// Mitsubishi GX Works2 project: JuiceProject221129   PLC: FX3G

// global labels: Global1
VAR_GLOBAL
  orange_stock AT D1106 : REAL;  (* רגיסטר מלאי תפוזים *)
  pomelo_stock AT D1108 : REAL;  (* רגיסטר מלאי פומלות *)
  clementine_stock AT D1110 : REAL;  (* רגיסטר מלאי קלמנטינות *)
  orange_washing AT D1112 : REAL;  (* רגיסטר מכונת שטיפה תפוזים *)
  pomelo_washing AT D1114 : REAL;  (* רגיסטר מכונת שטיפה פומלות *)
  clementine_washing AT D1116 : REAL;  (* רגיסטר מכונת שטיפה קלמנטינות *)
  squeeze_container AT D1124 : REAL;  (* מיכל סחיטה *)
  juice_container AT D1126 : REAL;  (* מיכל מיץ *)
  analog_input_2 AT D8281 : INT;  (* בדיקת איכות באמצעות ערך אנלוגי 2 *)
  storage_container AT D1128 : REAL;  (* מיכל אחסון *)
  start_wash_SW AT X002 : BOOL;  (* מתג תחילת תהליך השטיפה *)
  timer0 AT TC0 : BOOL;  (* טיימר הדלקת נורה *)
  var_time_0 AT D1130 : INT;  (* זמן הדלקת נורה לטיימר 0 *)
  start_light_help AT M0 : BOOL;  (* נורת עזר לתחילת טיימר הדלקת נורה *)
  timer0_ans AT TS0 : BOOL;  (* תשובה לטיימר 0 *)
  starter_wash_help AT M1 : BOOL;  (* נורת עזר המתחילה את תהליך הדלקת הנורה *)
  switch_2 AT X002 : BOOL;  (* מתג הפעלת שטיפת פירות *)
  light_5 AT Y005 : BOOL;  (* הדלקת נורה לתחילת השטיפה *)
  start_collect AT X001 : BOOL;  (* תחילת איסוף הפירות *)
  light_1 AT Y001 : BOOL;  (* נורת איסוף פירות *)
  start_sqeeze_help AT M3 : BOOL;  (* נורת עזר לתחילת שלב הסחיטה *)
END_VAR
VAR_GLOBAL CONSTANT
  const300 : INT := 30;  (* קבוע 3 שניות *)
END_VAR
VAR_GLOBAL
  start_func1_help AT M4 : BOOL;  (* מפעיל פונקציית שטיפה *)
  holder_m1 AT M1 : BOOL;  (* מפעיל פונקציית שטיפה *)
  start_sqeeze AT X011 : BOOL;  (* תחילת שלב הסחיטה *)
  counter1 AT CC1 : BOOL;  (* מונה לחיצות על X11 *)
END_VAR
VAR_GLOBAL CONSTANT
  var_count1 : INT := 2;  (* קבוע טיימר משתנה *)
END_VAR
VAR_GLOBAL
  counter1_ans AT CS1 : BOOL;  (* תשובה למונה 1 *)
  timer2_ans AT TS2 : BOOL;  (* תשובה למונה 2 *)
  helper_blink_cycle AT M5 : BOOL;  (* נורת עזר למעגל הבהוב *)
  timer4_ans AT TS4 : BOOL;  (* תשובה לטיימר 4 *)
END_VAR
VAR_GLOBAL CONSTANT
  const50 : INT := 50;  (* קבוע 5 שניות *)
END_VAR
VAR_GLOBAL
  light_blink_helper6 AT M6 : BOOL;  (* נורת עזר להבהוב 1 *)
  timer2 AT TC2 : BOOL;  (* מונה 2 *)
  timer3 AT TC3 : BOOL;  (* מונה 3 *)
  timer3_ans AT TS3 : BOOL;  (* תשובה למונה 3 *)
  light_blink_helper7 AT M7 : BOOL;  (* נורת עזר להבהוב 2 *)
  timer4 AT TC4 : BOOL;  (* טיימר 4 *)
  light_blink_helper8 AT M8 : BOOL;  (* נורת עזר להעברה למיכל המיץ *)
  start_QA AT X003 : BOOL;  (* תחילת בדיקת איכות *)
  start_QA_help AT M9 : BOOL;  (* נורת עזר לבדיקת איכות *)
END_VAR
VAR_GLOBAL CONSTANT
  min_value_QA : REAL := 1.0;  (* ערך מינמלי לבדיקת איכות *)
END_VAR
VAR_GLOBAL
  min_val_help AT M11 : BOOL;  (* נורת עזר לבדיקת מינימום *)
END_VAR
VAR_GLOBAL CONSTANT
  max_val1 : REAL := 5.0;  (* ערך מקסימלי לבדיקת איכות *)
END_VAR
VAR_GLOBAL
  max_val_help AT M12 : BOOL;  (* נורת עזר לבדיקת מקסימום *)
  QA_sample1 AT D1134 : REAL;  (* דגימת איכות לאחר המרה *)
  check_help AT M10 : BOOL;  (* נורת עזר להפעלת בדיקת איכות *)
  QA_sample AT D1132 : INT;  (* דגימת איכות *)
END_VAR
VAR_GLOBAL CONSTANT
  k_div : REAL := 404.5;  (* קבוע חלוקה *)
END_VAR
VAR_GLOBAL
  QA_correct AT M13 : BOOL;  (* נורת עזר לבדיקת מקסימום *)
  timer5 AT TC5 : BOOL;  (* טיימר 5 *)
END_VAR
VAR_GLOBAL CONSTANT
  const5 : INT := 5;  (* קבוע 5 שניות *)
END_VAR
VAR_GLOBAL
  timer5_ans AT TS5 : BOOL;  (* תשובה לטיי מר5 *)
  QA_light_helper14 AT M14 : BOOL;  (* נורת עזר להדלקת נורת איכות *)
  counter2 AT CC2 : BOOL;  (* מונה למספר בדיקות איכות באיטרציה *)
  counter2_ans AT CS2 : BOOL;  (* תשובה למונה 2 *)
  reset_light_help15 AT M15 : BOOL;  (* נורת עזר לאיפוס *)
END_VAR
VAR_GLOBAL CONSTANT
  const500 : INT := 50;  (* קבוע 5 שניות *)
END_VAR
VAR_GLOBAL
  holder_timer_QA AT M16 : BOOL;  (* נורת עזר להחזקת הטיימר לנורת בדיקת איכות *)
  light_4 AT Y004 : BOOL;  (* נורת בדיקת איכות *)
  finish_QA_help AT M17 : BOOL;  (* נורת עזר לאינדיקציה לסיום בדיקת איכות *)
  QA_failed_help AT M18 : BOOL;  (* נורת עזר לאינדיקציה לכשלון בדיקת האיכות *)
  switch_10_startDay AT X010 : BOOL;  (* מתג תחילת יום *)
  light_10_while_work AT Y010 : BOOL;  (* נורת יום עבודה פעיל *)
  finish_day19_help AT M19 : BOOL;  (* נורת עזר לאינדיקציה לסיום יום *)
END_VAR
VAR_GLOBAL CONSTANT
  const2 : REAL := 2.0;  (* קבוע 2 שנית *)
END_VAR
VAR_GLOBAL
  pomelo_right_help20 AT M20 : BOOL;  (* נורת עזר לעמידה בתנאי תחילת יום *)
  con_start_day_help21 AT M21 : BOOL;  (* נורת עזר לעמידה בתנאי תחילת יום *)
END_VAR
VAR_GLOBAL CONSTANT
  const100 : REAL := 100.0;  (* קבוע 100 *)
END_VAR
VAR_GLOBAL
  orange_allowed AT D1136 : REAL;  (* רגיסטר השומר כמה תפוזים ניקח באיטרציה *)
  clementine_allowed AT D1138 : REAL;  (* רגיסטר השומר כמה קלמנטיות ניקח באיטרציה *)
  switch_end_day7 AT X007 : BOOL;  (* מתג חירום לסיום יום עבודה *)
  finish_iteration_help AT M22 : BOOL;  (* נורת עזר לאינדיקציה לסיום איטרציה *)
  finish_iteration_help2 AT M23 : BOOL;  (* נורת עזר לאינדיקציה לסיום איטרציה *)
  inventory_ends AT M24 : BOOL;  (* נורת עזר לבדיקת מצב המלאי בסיום איטרציה *)
END_VAR
VAR_GLOBAL CONSTANT
  const0 : REAL;  (* קבוע 0 *)
END_VAR
VAR_GLOBAL
  start_blink_help_25 AT M25 : BOOL;  (* תחילת הבהוה נורות גנרי *)
  light_2 AT Y002 : BOOL;  (* נורת סחיטה Y2 *)
  light_3 AT Y003 : BOOL;  (* נורת סחיטה Y3 *)
  light_26_help AT M26 : BOOL;  (* נורת עזר להבהוב *)
  light_blink_end_help_26 AT M26 : BOOL;  (* נורת עזר להפעלת הבהוב סוף יום *)
  light_help_27 AT M27 : BOOL;  (* נורת עזר להפעלת הבהוב סוף יום *)
  temp AT X005 : BOOL;
  timer6 AT TC6 : BOOL;  (* טיימר 6 *)
  timer6_ans AT TS6 : BOOL;  (* תשובה לטיימר6 *)
  finish_iteration_forever_help AT M30 : BOOL;  (* טיימר הדלקת נורה *)
  rst_OA_help AT M28 : BOOL;  (* נורת עזר לאיפוס בדיקת איכות *)
  finish_rst_inv29 AT M29 : BOOL;  (* נורת עזר לאינדיקציה לסיום איפוס משתני מלאי סוף יום *)
  while_day_help31 AT M31 : BOOL;
  timer7 AT TC7 : BOOL;  (* טיימר הדלקת נורה *)
  Timer7_ans AT TS7 : BOOL;  (* תשובה למונה7 *)
  analog_output_2 AT D8282 : INT;  (* יציאת ערך אנלוגי 2 *)
END_VAR
VAR_GLOBAL CONSTANT
  const00 : INT;  (* קבוע 0 *)
END_VAR
VAR_GLOBAL
  helper_start_day_34 AT M34 : BOOL;  (* נורת עזר לאינדיקציה על סיום איפוס הרגיסטרים בתחילת יום *)
  orange_passed_help_35 AT M35 : BOOL;  (* נורת עזר לאינדיקציה על סיום איפוס הרגיסטרים בתחילת יום *)
  temp1000 AT M100 : BOOL;
  dounation_time_help32 AT M32 : BOOL;  (* נורת עזר לאינדיקציה לסיום יום *)
END_VAR
VAR_GLOBAL CONSTANT
  const_dounation : REAL := 300.0;  (* קבוע לגובה המלאי לצורך תרומה *)
END_VAR
VAR_GLOBAL
  dounation_allowed33 AT M33 : BOOL;  (* נורת עזר לאינדיקציה לביצוע תרומה *)
END_VAR
VAR_GLOBAL CONSTANT
  const_dounation_prec : REAL := 0.5;  (* קבוע אחוז התרומה *)
END_VAR
VAR_GLOBAL
  timer8 AT TC8 : BOOL;  (* טיימר הדלקת נורה *)
  timer8_ans AT TS8 : BOOL;  (* תשובה לטיימר סעיף יצירתי *)
  orange_full_stock AT D1100 : REAL;  (* רגיסטר מלאי תחילת יום תפוזים *)
  pomelo_full_stock AT D1102 : REAL;  (* רגיסטר מלאי תחילת יום פומלות *)
  clementine_full_stock AT D1104 : REAL;  (* רגיסטר מלאי תחילת יום קלמנטינות *)
  light7_dounation AT Y007 : BOOL;  (* נורת תרומה *)
  temp_36 AT M36 : BOOL;  (* נורת עזר לתרומה *)
  counter3 AT CC3 : BOOL;  (* מעיד על יום עבודה *)
  counter3_ans AT CS3 : BOOL;  (* תשובה למונה 3 *)
  temp37 AT M37 : BOOL;
  temp_38 AT M38 : BOOL;
END_VAR
VAR_GLOBAL CONSTANT
  resftyfty : BOOL := 1;  (* תשובה למונה 3 *)
END_VAR
VAR_GLOBAL
  analog_output_help AT D8282 : REAL;  (* יציאת ערך אנלוגי 2 *)
  timer9 AT TC9 : BOOL;  (* טיימר הדלקת נורה *)
  timer9_ans AT TS9 : BOOL;  (* טיימר הדלקת נורה *)
  clemantino_right_help40 AT M40 : BOOL;
  inventory_ends_help41 AT M41 : BOOL;  (* נורת עזר לסיום מלאי *)
  timer10 AT TC10 : BOOL;  (* טיימר הדלקת נורה *)
  Timer10_ans AT TS10 : BOOL;  (* תשובה למונה10 *)
  temp42 AT M42 : BOOL;
  finsh_collect_help AT M100 : BOOL;  (* נורת עזר לסיום איסוף *)
END_VAR

// task Task_01 (event TRUE, interval 0, priority 31): POU_01

PROGRAM POU_01
VAR
  TC5 : BOOL;  (* תשובה למונה 1 *)
END_VAR
(* structured ladder/FBD written out as ST: instructions are called as NAME(EN, inputs, outputs); _pN, _eN, _tN stand for wires *)
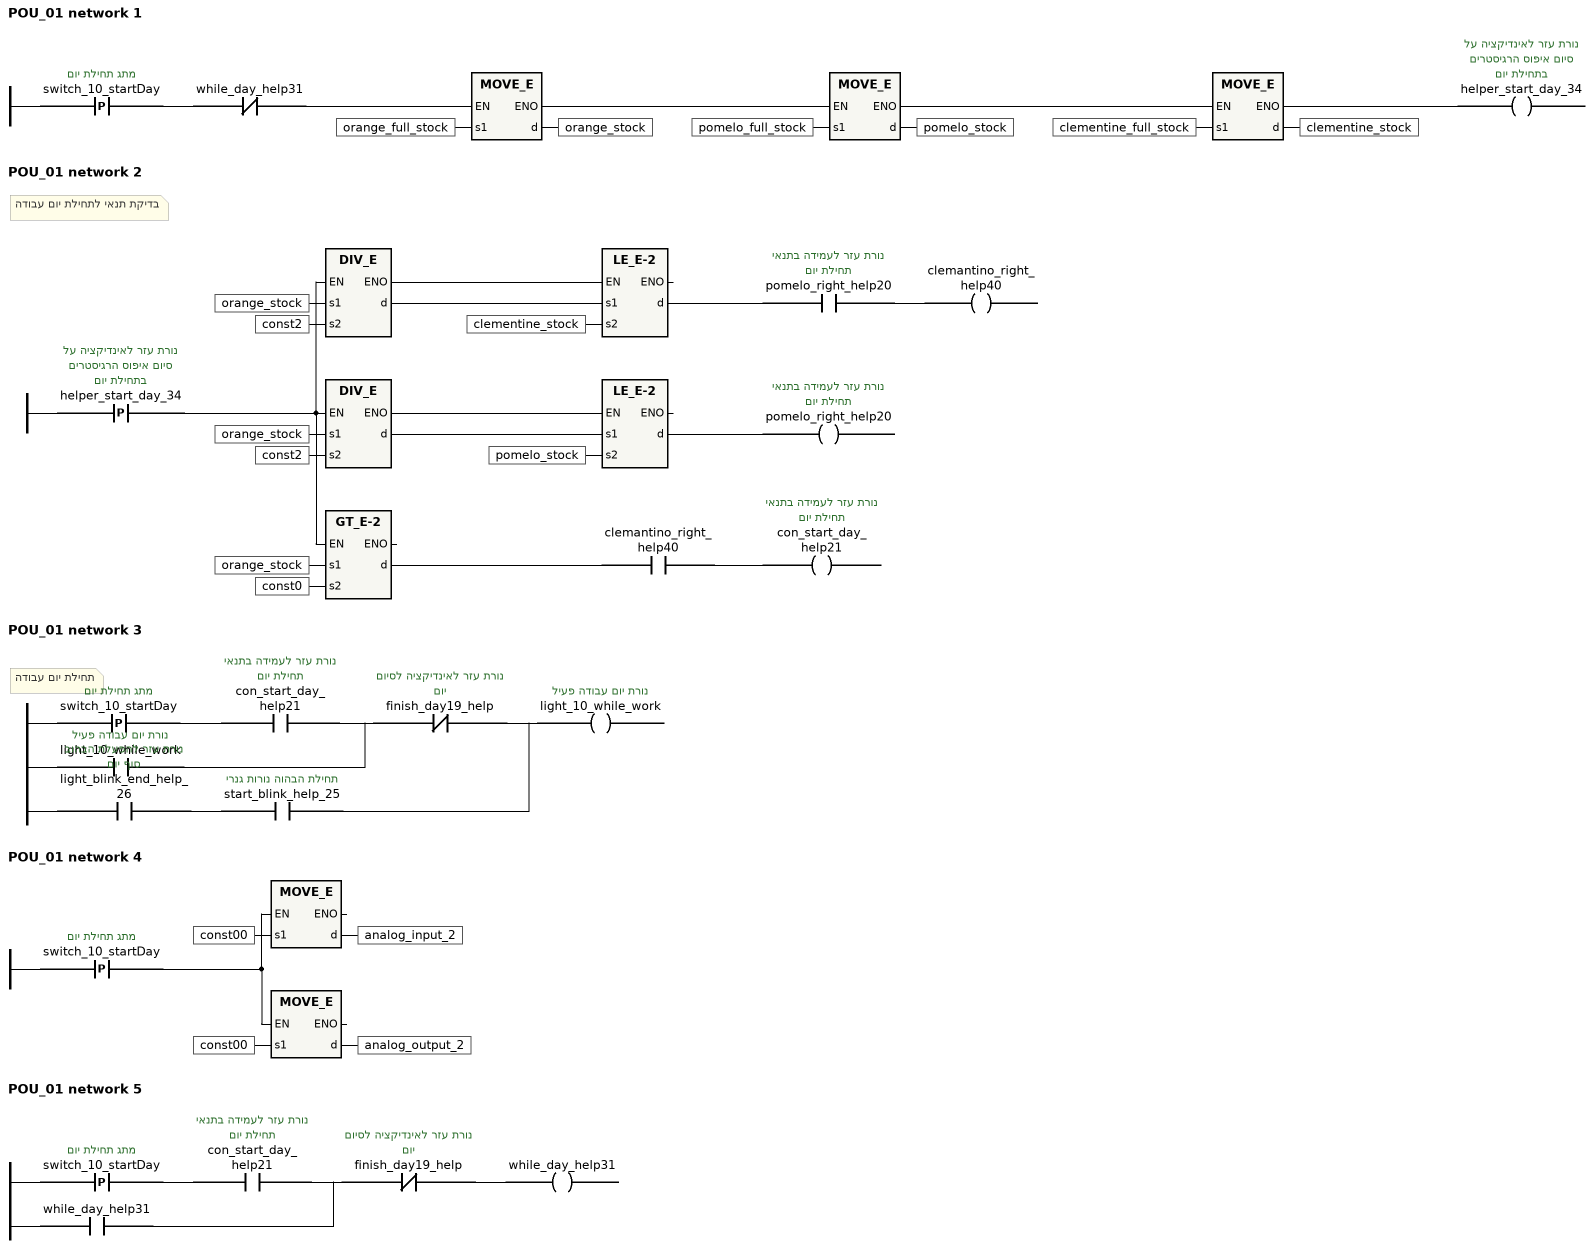
(* network 1 *)
_e1 := MOVE_E(LDP(TRUE, switch_10_startDay) AND NOT while_day_help31, orange_full_stock, orange_stock);
_e2 := MOVE_E(_e1, pomelo_full_stock, pomelo_stock);
_e3 := MOVE_E(_e2, clementine_full_stock, clementine_stock);
helper_start_day_34 := _e3;
(* network 2 *)
(* בדיקת תנאי לתחילת יום עבודה *)
_p1 := LDP(TRUE, helper_start_day_34);
_e3 := DIV_E(_p1, orange_stock, const2, _t2);
LE_E(_e3, _t2, pomelo_stock, _t4);
pomelo_right_help20 := _t4;
_e6 := DIV_E(_p1, orange_stock, const2, _t5);
LE_E(_e6, _t5, clementine_stock, _t7);
clemantino_right_help40 := _t7 AND pomelo_right_help20;
GT_E(_p1, orange_stock, const0, _t8);
con_start_day_help21 := _t8 AND clemantino_right_help40;
(* network 3 *)
(* תחילת יום עבודה *)
light_10_while_work := (((LDP(TRUE, switch_10_startDay) AND con_start_day_help21) OR light_10_while_work) AND NOT finish_day19_help) OR (light_blink_end_help_26 AND start_blink_help_25);
(* network 4 *)
_p1 := LDP(TRUE, switch_10_startDay);
MOVE_E(_p1, const00, analog_input_2);
MOVE_E(_p1, const00, analog_output_2);
(* network 5 *)
while_day_help31 := ((LDP(TRUE, switch_10_startDay) AND con_start_day_help21) OR while_day_help31) AND NOT finish_day19_help;
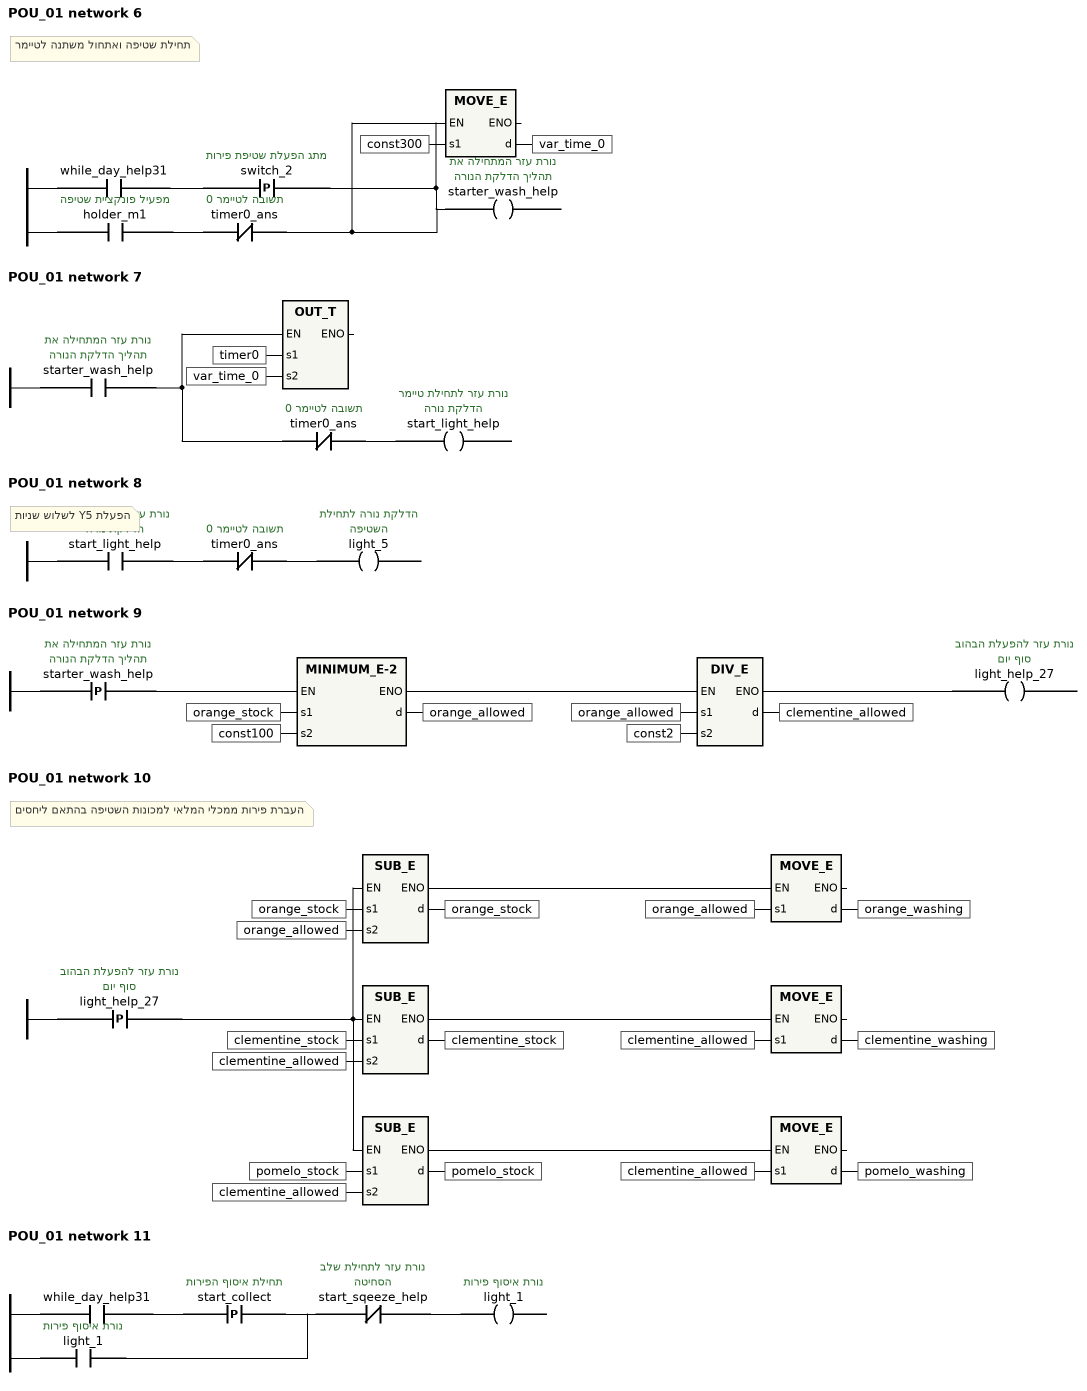
(* network 6 *)
(* תחילת שטיפה ואתחול משתנה לטיימר *)
_p1 := (while_day_help31 AND LDP(TRUE, switch_2)) OR (holder_m1 AND NOT timer0_ans);
MOVE_E(_p1, const300, var_time_0);
starter_wash_help := _p1;
(* network 7 *)
OUT_T(starter_wash_help, timer0, var_time_0);
start_light_help := starter_wash_help AND NOT timer0_ans;
(* network 8 *)
(* הפעלת Y5 לשלוש שניות *)
light_5 := start_light_help AND NOT timer0_ans;
(* network 9 *)
_e1 := MINIMUM_E(LDP(TRUE, starter_wash_help), orange_stock, const100, orange_allowed);
_e2 := DIV_E(_e1, orange_allowed, const2, clementine_allowed);
light_help_27 := _e2;
(* network 10 *)
(* העברת פירות ממכלי המלאי למכונות השטיפה בהתאם ליחסים *)
_p1 := LDP(TRUE, light_help_27);
_e2 := SUB_E(_p1, orange_stock, orange_allowed, orange_stock);
MOVE_E(_e2, orange_allowed, orange_washing);
_e3 := SUB_E(_p1, clementine_stock, clementine_allowed, clementine_stock);
MOVE_E(_e3, clementine_allowed, clementine_washing);
_e4 := SUB_E(_p1, pomelo_stock, clementine_allowed, pomelo_stock);
MOVE_E(_e4, clementine_allowed, pomelo_washing);
(* network 11 *)
light_1 := ((while_day_help31 AND LDP(TRUE, start_collect)) OR light_1) AND NOT start_sqeeze_help;
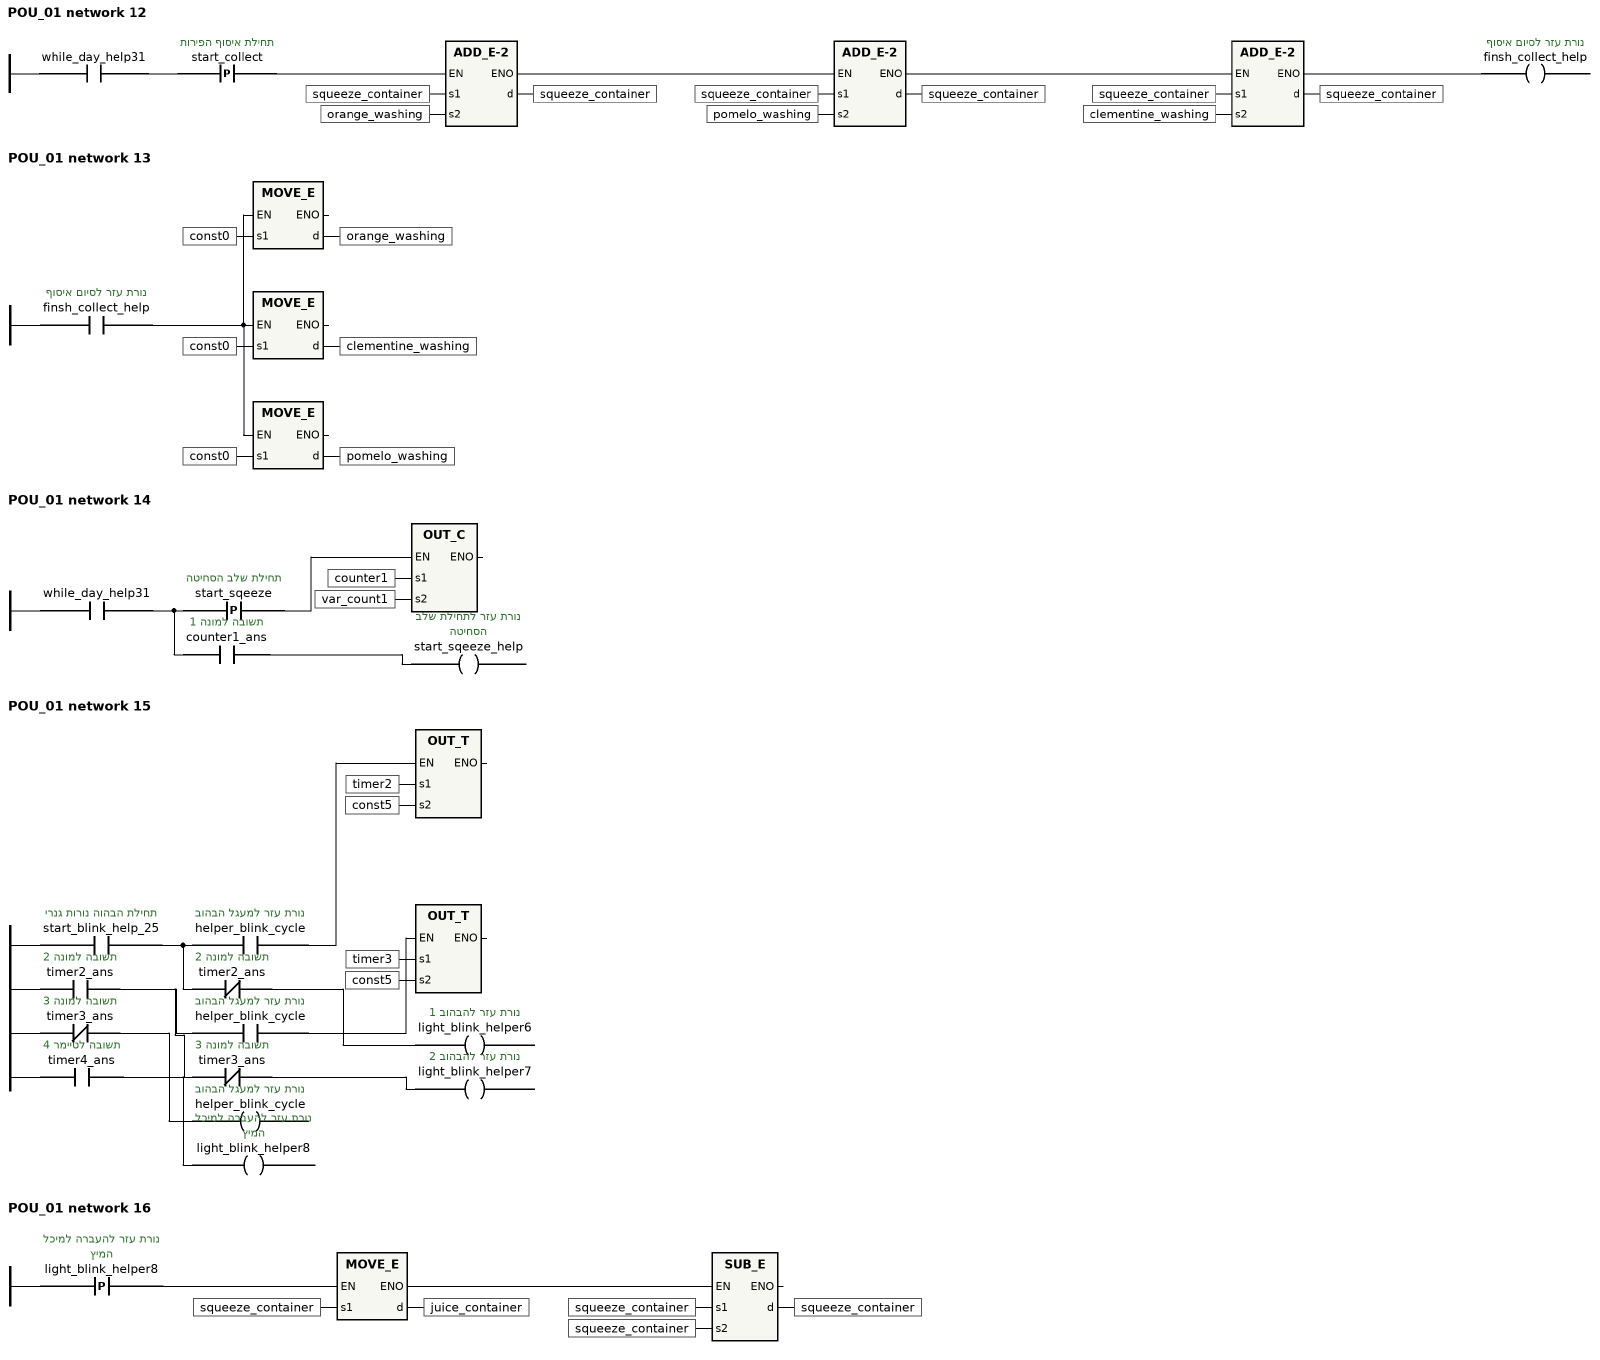
(* network 12 *)
_e1 := ADD_E(while_day_help31 AND LDP(TRUE, start_collect), squeeze_container, orange_washing, squeeze_container);
_e2 := ADD_E(_e1, squeeze_container, pomelo_washing, squeeze_container);
_e3 := ADD_E(_e2, squeeze_container, clementine_washing, squeeze_container);
finsh_collect_help := _e3;
(* network 13 *)
MOVE_E(finsh_collect_help, const0, orange_washing);
MOVE_E(finsh_collect_help, const0, clementine_washing);
MOVE_E(finsh_collect_help, const0, pomelo_washing);
(* network 14 *)
OUT_C(while_day_help31 AND LDP(TRUE, start_sqeeze), counter1, var_count1);
start_sqeeze_help := while_day_help31 AND counter1_ans;
(* network 15 *)
OUT_T(start_blink_help_25 AND helper_blink_cycle, timer2, const5);
light_blink_helper6 := start_blink_help_25 AND NOT timer2_ans;
OUT_T(timer2_ans AND helper_blink_cycle, timer3, const5);
light_blink_helper7 := timer2_ans AND NOT timer3_ans;
helper_blink_cycle := NOT timer3_ans;
light_blink_helper8 := timer4_ans;
(* network 16 *)
_e1 := MOVE_E(LDP(TRUE, light_blink_helper8), squeeze_container, juice_container);
SUB_E(_e1, squeeze_container, squeeze_container, squeeze_container);
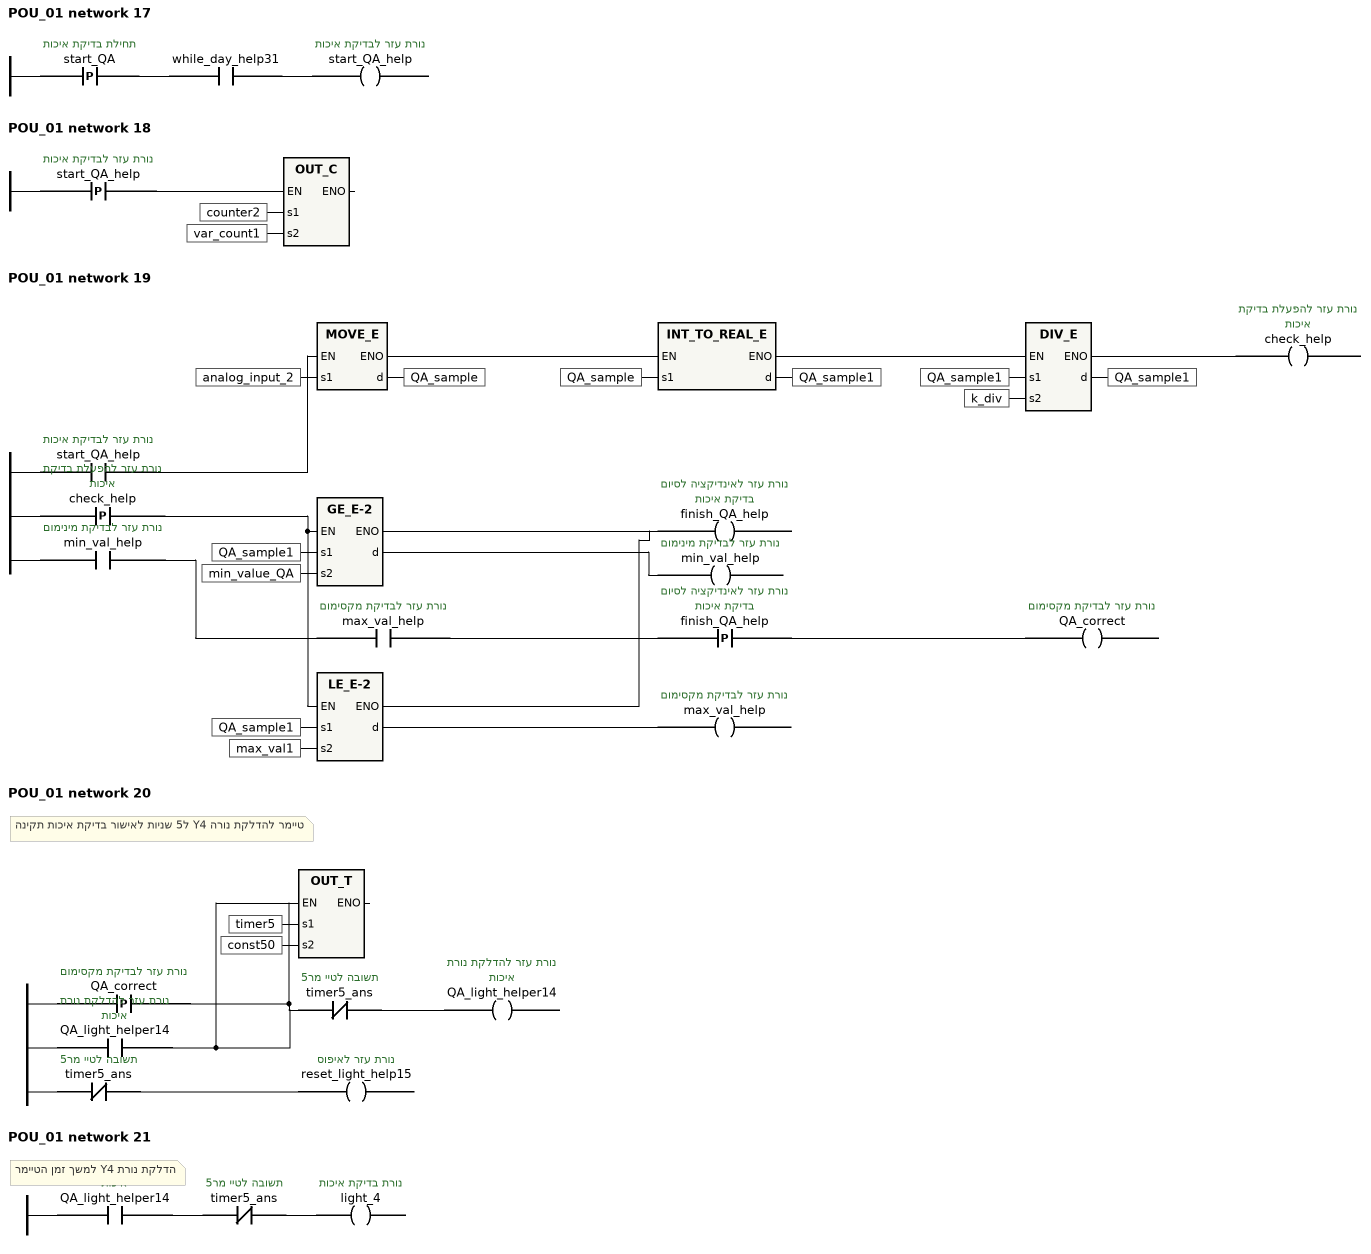
(* network 17 *)
start_QA_help := LDP(TRUE, start_QA) AND while_day_help31;
(* network 18 *)
OUT_C(LDP(TRUE, start_QA_help), counter2, var_count1);
(* network 19 *)
_e1 := MOVE_E(start_QA_help, analog_input_2, QA_sample);
_e2 := INT_TO_REAL_E(_e1, QA_sample, QA_sample1);
_e3 := DIV_E(_e2, QA_sample1, k_div, QA_sample1);
check_help := _e3;
_p4 := LDP(TRUE, check_help);
_e6 := GE_E(_p4, QA_sample1, min_value_QA, _t5);
_e8 := LE_E(_p4, QA_sample1, max_val1, _t7);
finish_QA_help := _e6 OR _e8;
min_val_help := _t5;
max_val_help := _t7;
QA_correct := min_val_help AND max_val_help AND LDP(TRUE, finish_QA_help);
(* network 20 *)
(* טיימר להדלקת נורה Y4 ל5 שניות לאישור בדיקת איכות תקינה *)
_p1 := LDP(TRUE, QA_correct) OR QA_light_helper14;
OUT_T(_p1, timer5, const50);
QA_light_helper14 := _p1 AND NOT timer5_ans;
reset_light_help15 := NOT timer5_ans;
(* network 21 *)
(* הדלקת נורת Y4 למשך זמן הטיימר *)
light_4 := QA_light_helper14 AND NOT timer5_ans;
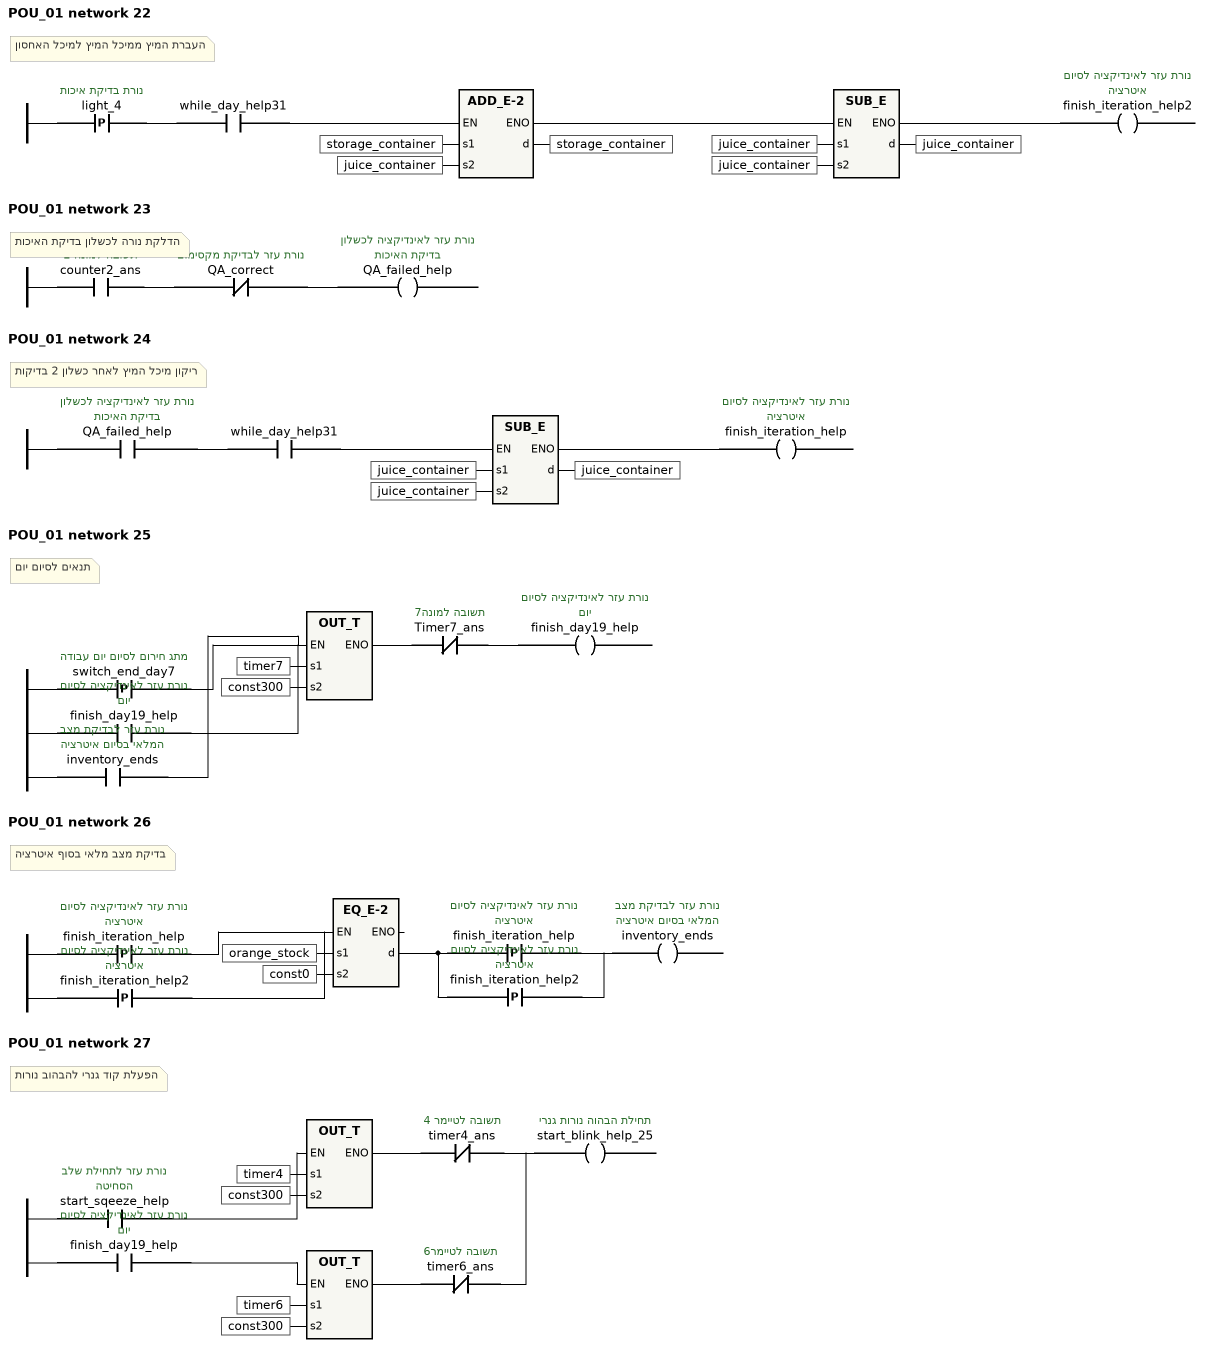
(* network 22 *)
(* העברת המיץ ממיכל המיץ למיכל האחסון *)
_e1 := ADD_E(LDP(TRUE, light_4) AND while_day_help31, storage_container, juice_container, storage_container);
_e2 := SUB_E(_e1, juice_container, juice_container, juice_container);
finish_iteration_help2 := _e2;
(* network 23 *)
(* הדלקת נורה לכשלון בדיקת האיכות *)
QA_failed_help := counter2_ans AND NOT QA_correct;
(* network 24 *)
(* ריקון מיכל המיץ לאחר כשלון 2 בדיקות *)
_e1 := SUB_E(QA_failed_help AND while_day_help31, juice_container, juice_container, juice_container);
finish_iteration_help := _e1;
(* network 25 *)
(* תנאים לסיום יום *)
_e1 := OUT_T(LDP(TRUE, switch_end_day7) OR finish_day19_help OR inventory_ends, timer7, const300);
finish_day19_help := _e1 AND NOT Timer7_ans;
(* network 26 *)
(* בדיקת מצב מלאי בסוף איטרציה *)
EQ_E(LDP(TRUE, finish_iteration_help) OR LDP(TRUE, finish_iteration_help2), orange_stock, const0, _t1);
inventory_ends := (_t1 AND LDP(TRUE, finish_iteration_help)) OR (_t1 AND LDP(TRUE, finish_iteration_help2));
(* network 27 *)
(* הפעלת קוד גנרי להבהוב נורות *)
_e1 := OUT_T(start_sqeeze_help, timer4, const300);
_e2 := OUT_T(finish_day19_help, timer6, const300);
start_blink_help_25 := (_e1 AND NOT timer4_ans) OR (_e2 AND NOT timer6_ans);
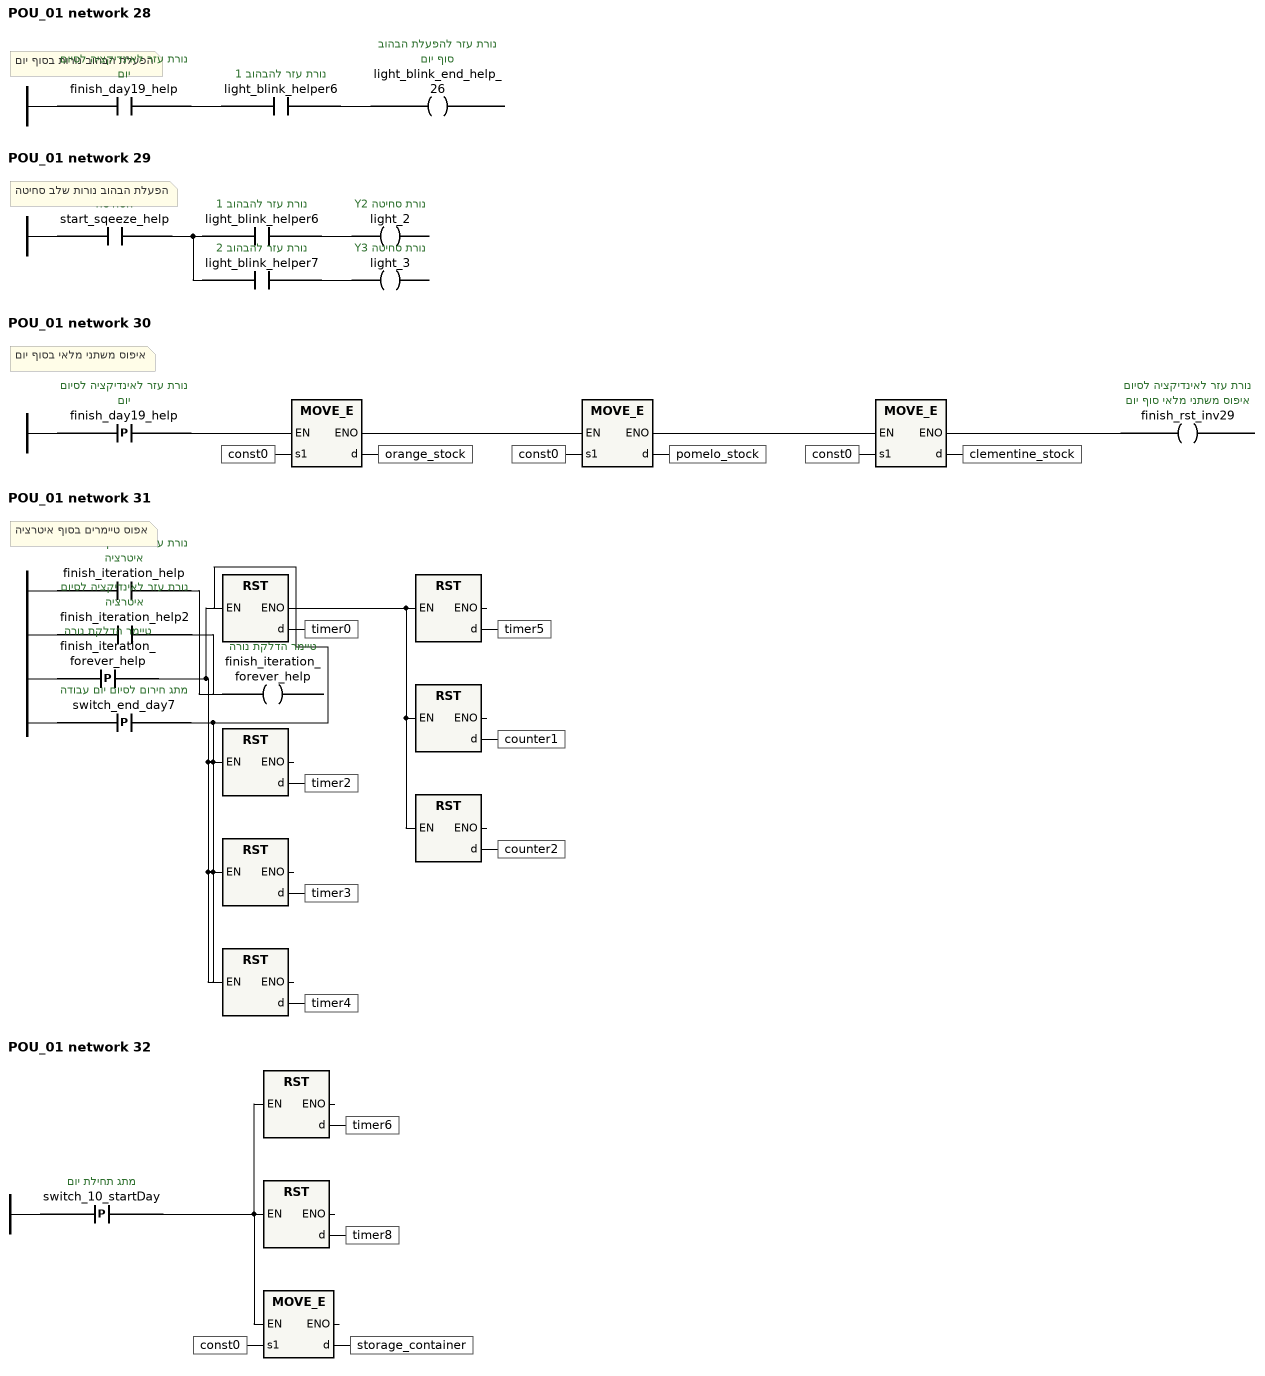
(* network 28 *)
(* הפעלת הבהוב נורות בסוף יום *)
light_blink_end_help_26 := finish_day19_help AND light_blink_helper6;
(* network 29 *)
(* הפעלת הבהוב נורות שלב סחיטה *)
light_2 := start_sqeeze_help AND light_blink_helper6;
light_3 := start_sqeeze_help AND light_blink_helper7;
(* network 30 *)
(* איפוס משתני מלאי בסוף יום *)
_e1 := MOVE_E(LDP(TRUE, finish_day19_help), const0, orange_stock);
_e2 := MOVE_E(_e1, const0, pomelo_stock);
_e3 := MOVE_E(_e2, const0, clementine_stock);
finish_rst_inv29 := _e3;
(* network 31 *)
(* אפוס טיימרים בסוף איטרציה *)
finish_iteration_forever_help := finish_iteration_help OR finish_iteration_help2;
_p1 := LDP(TRUE, finish_iteration_forever_help) OR LDP(TRUE, switch_end_day7);
_e2 := RST(_p1, timer0);
RST(_e2, timer5);
RST(_p1, timer2);
RST(_p1, timer3);
RST(_e2, counter1);
RST(_p1, timer4);
RST(_e2, counter2);
(* network 32 *)
_p1 := LDP(TRUE, switch_10_startDay);
RST(_p1, timer6);
RST(_p1, timer8);
MOVE_E(_p1, const0, storage_container);
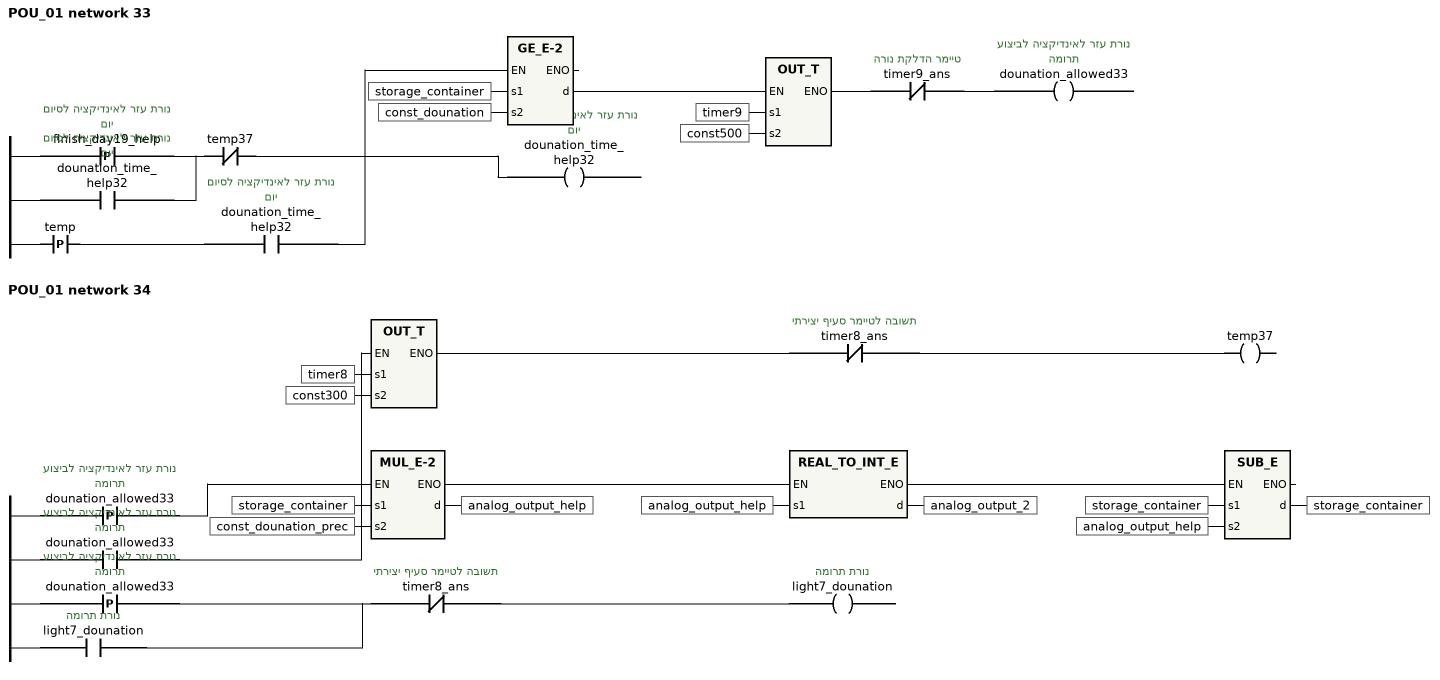
(* network 33 *)
dounation_time_help32 := (LDP(TRUE, finish_day19_help) OR dounation_time_help32) AND NOT temp37;
GE_E(LDP(TRUE, temp) AND dounation_time_help32, storage_container, const_dounation, _t1);
_e2 := OUT_T(_t1, timer9, const500);
dounation_allowed33 := _e2 AND NOT timer9_ans;
(* network 34 *)
_e1 := MUL_E(LDP(TRUE, dounation_allowed33), storage_container, const_dounation_prec, analog_output_help);
_e2 := OUT_T(dounation_allowed33, timer8, const300);
temp37 := _e2 AND NOT timer8_ans;
_e3 := REAL_TO_INT_E(_e1, analog_output_help, analog_output_2);
SUB_E(_e3, storage_container, analog_output_help, storage_container);
light7_dounation := (LDP(TRUE, dounation_allowed33) OR light7_dounation) AND NOT timer8_ans;
END_PROGRAM
